(* IEC 61131-3 sources: remote-repo/src, 4 files *)

(* ---- SpeedAxis.st ---- *)
USING Siemens.Simatic.S71500.MotionControl.Native;

NAMESPACE TiaProject.Direct_loading_TIADemo
    TYPE
        MotionCommand : STRUCT
            enableAxis : BOOL;
            reset : BOOL;
            jogForward : BOOL;
            jogBackward : BOOL;
            velocitySetpoint : LREAL :=300.0;
            actualSpeed : LREAL;
        END_STRUCT;

    END_TYPE

    CLASS SpeedAxisControl

        VAR PUBLIC
            AxisCommand : REF_TO MotionCommand;
        END_VAR

        VAR
            //initialization button
            IsInitialized : BOOL;
            //to object
            SpeedAxis : REF_TO TO_SpeedAxis;
            //instances for MC instructions
            _instPower : MC_Power;
            _instReset : MC_Reset;
            _instJog : MC_MoveJog;
        END_VAR

        METHOD PUBLIC Initialize
            VAR_INPUT
                _speedAxisRef : REF_TO TO_SpeedAxis;
            END_VAR
            IF IsInitialized THEN
                RETURN;
            ELSIF _speedAxisRef<> NULL THEN
                SpeedAxis := _speedAxisRef;
                IsInitialized := TRUE;
            END_IF;
        END_METHOD

        METHOD PUBLIC Execute
            //power on axis
            _instPower(Axis:=SpeedAxis^,enable:=AxisCommand^.enableAxis);
            //jog axis
            _instJog(Axis:=SpeedAxis^,JogForward := AxisCommand^.jogForward,
            JogBackward := AxisCommand^.jogBackward,velocity:=AxisCommand^.velocitySetpoint);
            //reset axis
            _instReset(Axis:=SpeedAxis^,Execute:=AxisCommand^.reset);
            //read actual speed
            AxisCommand^.actualSpeed := SpeedAxis^.Velocity;
        END_METHOD
    END_CLASS
END_NAMESPACE

(* ---- FB.st ---- *)
FUNCTION_BLOCK FB
    VAR_IN_OUT
        arr1: ARRAY [0..9] OF INT; // 假设我们有一个包含10个整数的数组
        arr2: ARRAY [0..9] OF INT;
    END_VAR

    VAR
       variable : INT;
    END_VAR
      // 初始化数组示例
    VAR_TEMP
        index : INT;
        shiftIndex : INT;
        index_j : INT;
        temp: INT;               // 临时变量
    END_VAR

    // 比较两个数组中是否有相同的元素，有的话把相同元素提取出来
        FOR index := 0 TO 9 DO
            FOR shiftIndex := 0 TO 9 DO
                IF arr1[index] = arr2[shiftIndex] THEN
                    // 找到相同的元素，提取出来
                    temp := arr1[index];
                    FOR index_j := index TO 8 DO
                        arr1[index_j] := arr1[index_j+1];
                    END_FOR;
                    arr1[9] := 0; // 将最后一个元素设置为0
                END_IF;
            END_FOR;
        END_FOR;

        // 将提取出来的元素赋值给变量
        variable := temp;

END_FUNCTION_BLOCK

(* ---- configuration.st ---- *)
USING TiaProject.Direct_loading_TIADemo;
CONFIGURATION MyConfiguration
    TASK Main(Priority := 1);

    PROGRAM P1 WITH Main: MainProgram;

    VAR_GLOBAL
       speedAxisInstance : SpeedAxisControl:=(AxisCommand:=REF(PosAxisCommand));
       PosAxisCommand : MotionCommand;
    END_VAR
END_CONFIGURATION

(* ---- MainProgram.st ---- *)
USING TiaProject.Direct_loading_TIADemo;
USING Siemens.Simatic.S71500.MotionControl.Native;
PROGRAM MainProgram
    VAR_EXTERNAL
        speedAxisInstance : TiaProject.Direct_loading_TIADemo.SpeedAxisControl;
        PosAxisCommand : TiaProject.Direct_loading_TIADemo.MotionCommand;
    END_VAR

    VAR
        _SpeedAxis : DB_ANY := UINT#1;
    END_VAR

    speedAxisInstance.Initialize(AsSpeedAxisRef(_SpeedAxis));
    speedAxisInstance.Execute();
    ;
END_PROGRAM
